INTERFACE I_ChunkedResponseData EXTENDS I_SessionData

PROPERTY PUBLIC SendComplete : BOOL
GET
END_GET
END_PROPERTY

METHOD PUBLIC SendNextChunk
VAR_INPUT
	Response : I_ServerResponse;
	Size : UDINT;
END_VAR
END_METHOD

PROPERTY SizeRemaining : UDINT
GET
END_GET
END_PROPERTY

END_INTERFACE

(* stored: Version 1.1.0.1, ProductVersion 3.1.4024.12
   Itf I_ChunkedResponseData: Id {69610c76-4c21-08d1-2052-c6a6d5230283}
   Property SendComplete: Id {89c22128-d662-0889-10f1-aa9df2af4a6c}
   Get Get: Id {35ce893f-d97d-0dab-0646-4fced105dcd4}
   Method SendNextChunk: Id {2b9eeb99-2fdb-0b43-26b8-71132cec4ed7}
   Property SizeRemaining: Id {bac0b717-a761-029c-3f5e-e54d3e3f4141}
   Get Get: Id {a1453d97-1bc6-053d-1d1a-1b85b3ae579f} *)
